// TIA Portal V17 export
// export: Created 2024-08-26T21:10:49.0758325Z, ExportSetting WithDefaults, DisplayName Totally Integrated Automation Portal, DisplayVersion V17 Update 7, DisplayName TIA Portal Openness, DisplayVersion V17 Update 7, DisplayName TIA Portal Version Control Interface, DisplayVersion V17, DisplayName SINAMICS Startdrive Advanced, DisplayVersion V17 SP2, DisplayName SINAMICS Startdrive G110M, G120, G120C, G120D, G120P, G115D, DisplayVersion V17 SP2, DisplayName SINAMICS Startdrive G130, G150, S120, S150, SINAMICS MV, S210, DisplayVersion V17 SP2, DisplayName STEP 7 Professional, DisplayVersion V17 Update 7, DisplayName STEP 7 Safety, DisplayVersion V17 Update 6, DisplayName WinCC Advanced / Unified PC, DisplayVersion V17 Update 7
FUNCTION_BLOCK "CODE READING"   // FB13, LAD
{ S7_Optimized_Access := 'TRUE' }
VERSION : 0.1
// stored: AutoNumber true, IsIECCheckEnabled false, IsRetainMemResEnabled false, MemoryReserve 100, SetENOAutomatically false, UDAEnableTagReadback false
   VAR_INPUT
      hwAdd : HW_IO;
      scannerBusy : Bool;
      autoMode : Bool;
      manualMode : Bool;
      scannerReadingComplete : Bool;
      scannerReadingError : Bool;
      clearData : Bool;
      scannerDataSize : Int;
      requestScannerAuto : Bool;
      requestScannerManual : Bool;
      scannerEnabled : Bool;
      labelIdentyfier : String[5];
      labelPosition : Int;
      labelIdentyfier_2 : String[5];
      labelPosition_2 : Int;
      label1 : Bool;
      label2 : Bool;
   END_VAR
   VAR_OUTPUT
      hmiLabel : String[180];
      scannerOk : Bool;
      scannerOk_2 : Bool;
      clearReadComplete : Bool;
      requestScannerOutput : Bool;
      codeRead : Bool;
   END_VAR
   VAR
      scannerReading { ExternalAccessible := 'False'; ExternalVisible := 'False'; ExternalWritable := 'False'} : Array[0..254] of Char;
      ScannerReadTimer { S7_SetPoint := 'True'} : TON_TIME;
   END_VAR
   VAR_TEMP
      scannerError : Int;
      receiveCode : String[80];
      readingScann1 : String[180];
      scannerLength : Int;
      labelExtract : String[10];
   END_VAR
   VAR_TEMP   // added for the SCL form of the ladder/FBD networks
      _w1 : Bool;
      _w2 : Bool;
      _w3 : Bool;
      _w4 : Bool;
      _w5 : Bool;
      _w6 : Bool;
      _w7 : Bool;
      _w8 : Bool;
      _w9 : Bool;
      _w10 : Bool;
      _w11 : Bool;
   END_VAR
BEGIN

REGION Network 1: REQUEST SCANNER
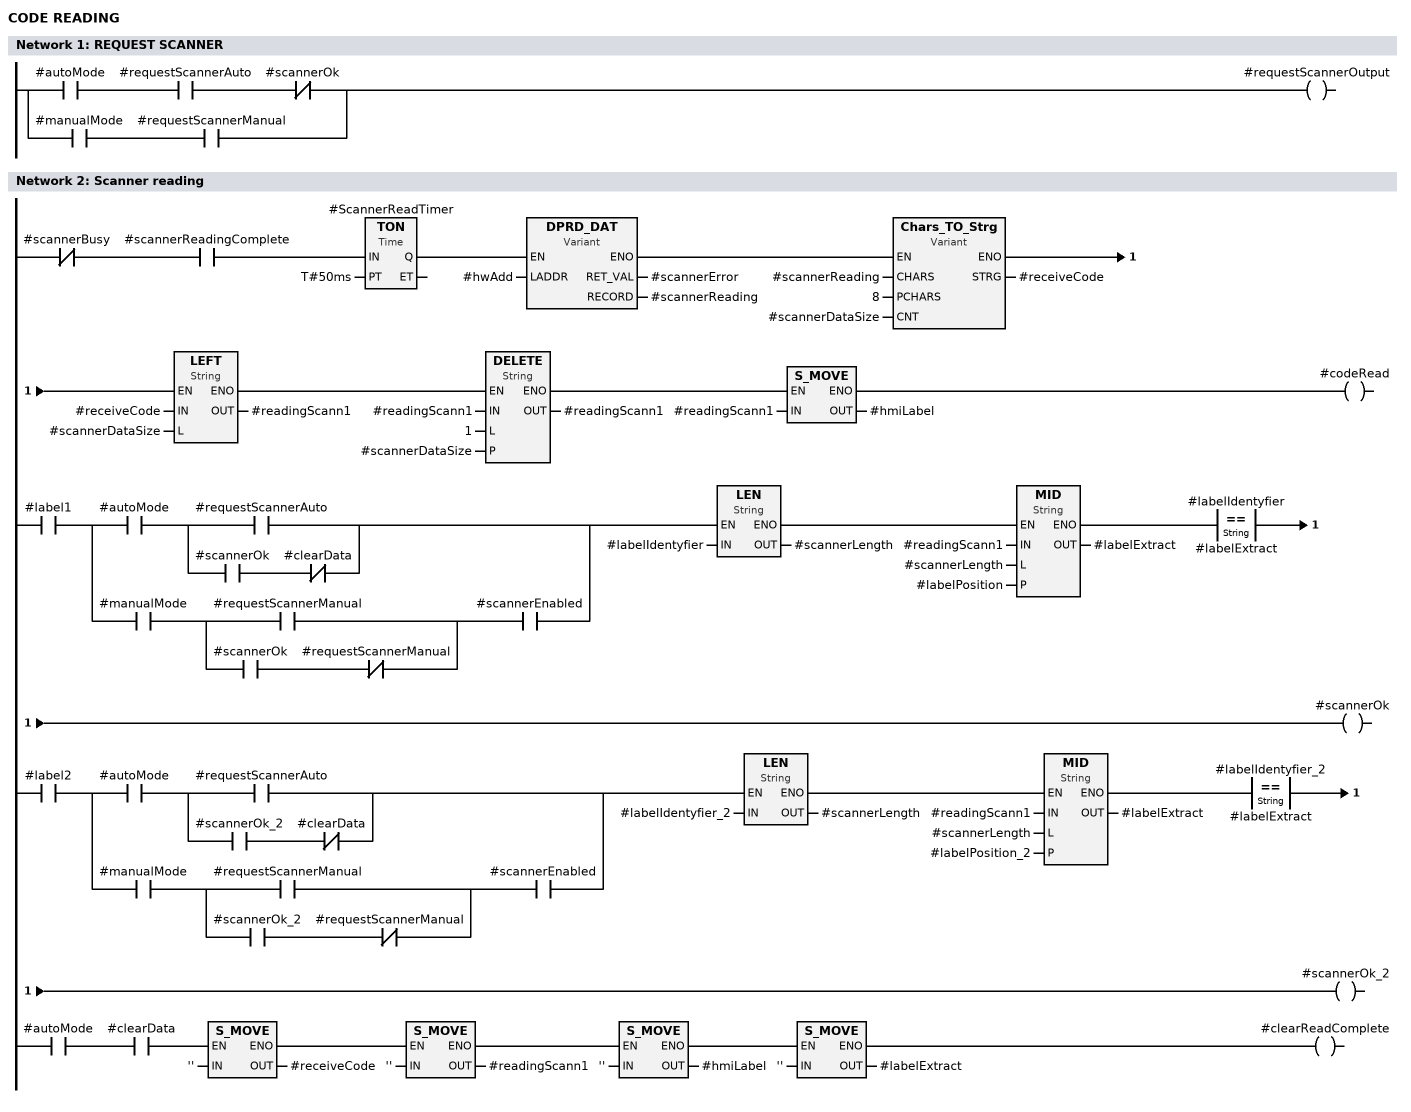
   RUNG wire#powerrail
      Contact( #autoMode )
      Contact( #requestScannerAuto )
      I_Contact( #scannerOk )
      wire#w1
      Coil( #requestScannerOutput )
   END_RUNG
   RUNG wire#powerrail
      Contact( #manualMode )
      Contact( #requestScannerManual )
   END_RUNG wire#w1
   // the same network as SCL:
   #requestScannerOutput := (#autoMode AND #requestScannerAuto AND NOT #scannerOk) OR (#manualMode AND #requestScannerManual);
END_REGION

REGION Network 2: Scanner reading
   RUNG wire#powerrail
      I_Contact( #scannerBusy )
      Contact( #scannerReadingComplete )
      { S7_Templates := "time_type := Time" } #ScannerReadTimer.TON(pt := T#50ms, et =>)
      { S7_Templates := "[ptr_type := Variant, laddr_type := HW_IO]" } DPRD_DAT(LADDR := #hwAdd, RET_VAL => #scannerError, RECORD => #scannerReading)
      { S7_Templates := "[ptr_type := Variant, str_type := String]" } Chars_TO_Strg(Chars := #scannerReading, pChars := 8, Cnt := #scannerDataSize, Strg => #receiveCode)
      { S7_Templates := "str_type := String" } LEFT(IN := #receiveCode, L := #scannerDataSize, OUT => #readingScann1)
      { S7_Templates := "str_type := String" } DELETE(IN := #readingScann1, L := 1, P := #scannerDataSize, OUT => #readingScann1)
      S_Move(in := #readingScann1, out => #hmiLabel)
      Coil( #codeRead )
   END_RUNG
   RUNG wire#powerrail
      Contact( #label1 )
      wire#w1
      Contact( #autoMode )
      wire#w2
      Contact( #requestScannerAuto )
      wire#w3
      { S7_Templates := "[str_type := String, return_type := Int]" } LEN(IN := #labelIdentyfier, OUT => #scannerLength)
      { S7_Templates := "value_type := String" } MID(IN := #readingScann1, L := #scannerLength, P := #labelPosition, OUT => #labelExtract)
      { S7_Templates := "SrcType := String" } EQ_Contact(in1 := #labelIdentyfier, in2 := #labelExtract)
      Coil( #scannerOk )
   END_RUNG
   RUNG wire#w2
      Contact( #scannerOk )
      I_Contact( #clearData )
   END_RUNG wire#w3
   RUNG wire#w1
      Contact( #manualMode )
      wire#w4
      Contact( #requestScannerManual )
      wire#w5
      Contact( #scannerEnabled )
   END_RUNG wire#w3
   RUNG wire#w4
      Contact( #scannerOk )
      I_Contact( #requestScannerManual )
   END_RUNG wire#w5
   RUNG wire#powerrail
      Contact( #label2 )
      wire#w6
      Contact( #autoMode )
      wire#w7
      Contact( #requestScannerAuto )
      wire#w8
      { S7_Templates := "[str_type := String, return_type := Int]" } LEN(IN := #labelIdentyfier_2, OUT => #scannerLength)
      { S7_Templates := "value_type := String" } MID(IN := #readingScann1, L := #scannerLength, P := #labelPosition_2, OUT => #labelExtract)
      { S7_Templates := "SrcType := String" } EQ_Contact(in1 := #labelIdentyfier_2, in2 := #labelExtract)
      Coil( #scannerOk_2 )
   END_RUNG
   RUNG wire#w7
      Contact( #scannerOk_2 )
      I_Contact( #clearData )
   END_RUNG wire#w8
   RUNG wire#w6
      Contact( #manualMode )
      wire#w9
      Contact( #requestScannerManual )
      wire#w10
      Contact( #scannerEnabled )
   END_RUNG wire#w8
   RUNG wire#w9
      Contact( #scannerOk_2 )
      I_Contact( #requestScannerManual )
   END_RUNG wire#w10
   RUNG wire#powerrail
      Contact( #autoMode )
      Contact( #clearData )
      S_Move(in := '', out => #receiveCode)
      S_Move(in := '', out => #readingScann1)
      S_Move(in := '', out => #hmiLabel)
      S_Move(in := '', out => #labelExtract)
      Coil( #clearReadComplete )
   END_RUNG
   // the same network as SCL:
   #ScannerReadTimer(IN := NOT #scannerBusy AND #scannerReadingComplete, PT := T#50ms);   // TON
   #scannerError := DPRD_DAT(EN := #ScannerReadTimer.Q, LADDR := #hwAdd, RECORD => #scannerReading, ENO => #_w1);
   Chars_TO_Strg(EN := #_w1,
                 Chars := #scannerReading,
                 pChars := 8,
                 Cnt := #scannerDataSize,
                 Strg => #receiveCode,
                 ENO => #_w2);
   LEFT(EN := #_w2, IN := #receiveCode, L := #scannerDataSize, OUT => #readingScann1, ENO => #_w3);
   DELETE(EN := #_w3, IN := #readingScann1, L := 1, P := #scannerDataSize, OUT => #readingScann1, ENO => #_w4);
   IF #_w4 THEN #hmiLabel := #readingScann1; END_IF;
   #codeRead := #_w4;
   #_w5 := #label1 AND ((#autoMode AND (#requestScannerAuto OR (#scannerOk AND NOT #clearData))) OR (#manualMode AND (#requestScannerManual OR (#scannerOk AND NOT #requestScannerManual)) AND #scannerEnabled));
   LEN(EN := #_w5, IN := #labelIdentyfier, OUT => #scannerLength, ENO => #_w6);
   MID(EN := #_w6,
       IN := #readingScann1,
       L := #scannerLength,
       P := #labelPosition,
       OUT => #labelExtract,
       ENO => #_w7);
   #scannerOk := #_w7 AND (#labelIdentyfier = #labelExtract);
   #_w8 := #label2 AND ((#autoMode AND (#requestScannerAuto OR (#scannerOk_2 AND NOT #clearData))) OR (#manualMode AND (#requestScannerManual OR (#scannerOk_2 AND NOT #requestScannerManual)) AND #scannerEnabled));
   LEN(EN := #_w8, IN := #labelIdentyfier_2, OUT => #scannerLength, ENO => #_w9);
   MID(EN := #_w9,
       IN := #readingScann1,
       L := #scannerLength,
       P := #labelPosition_2,
       OUT => #labelExtract,
       ENO => #_w10);
   #scannerOk_2 := #_w10 AND (#labelIdentyfier_2 = #labelExtract);
   #_w11 := #autoMode AND #clearData;
   IF #_w11 THEN
       #receiveCode := '';
       #readingScann1 := '';
       #hmiLabel := '';
       #labelExtract := '';
   END_IF;
   #clearReadComplete := #_w11;
END_REGION
END_FUNCTION_BLOCK
